VAR_GLOBAL
		stDutData_Cnc3					: ST_Dut_Data;
END_VAR

(* stored: Version 1.1.0.1, ProductVersion 3.1.4024.12
   GVL GVL_CNC3: Id {15f86b19-9643-4e1e-ba21-f63db974a140} *)
